// TIA Portal V17 export
// export: Created 2025-06-26T07:49:55.7582925Z, ExportSetting WithDefaults, DisplayName Totally Integrated Automation Portal, DisplayVersion V17 Update 8, DisplayName TIA Portal Openness, DisplayVersion V17 Update 8, DisplayName TIA Portal Version Control Interface, DisplayVersion V17, DisplayName STEP 7 Professional, DisplayVersion V17 Update 8, DisplayName STEP 7 Safety, DisplayVersion V17 Update 6, DisplayName WinCC Advanced, DisplayVersion V17 Update 8
TYPE "stPID_Regulator"
// stored: IsFailsafeCompliant false
   STRUCT
      fControlDeviation : Real;   // Deviation = SP - PV
      fOutMax : Real;
      fOutMin : Real;
      fOut : Real;   // Manipulated value
      bManualMode : Bool;   // 1 = manual mode, 0 = auto
      fManualValue : Real;
      Kp : Real;   // Proportional gain
      Tn : Real;   // Integral gain (reset time)
      Tv : Real;   // Velocity or derivative gain
      T1 : Real;   // Differentiator smoothing factor
      bAtMin : Bool;   // Controller negative saturation
      bAtMax : Bool;   // Controller positive saturation
   END_STRUCT;
END_TYPE
